(* Logix 5000 project; controller Safety vendor 1 type 14 code 148 rev 32.11; software revision 32.03; part 9 of 17 *)
(* tags used below, declared in another part *)
   DPD_EstopRstCmd : BOOL;   // DPD Estop Reset Cmd
   DPD_FltRstCmd : BOOL;   // DPD Fault Reset Cmd
   DPD_No_EStops : BOOL;   // DPD No Estops ( 1= OK)
   ESTOP_x281PB040 : DCI_STOP;   // OS9 Line EStop Pushbutton
   ESTOP_x281PB040_Flt : ALIAS FOR Flt_Estops.8;   // OS9 Line EStop Pushbutton Fault ( 1= Fault)
   ESTOP_x291PB040 : DCI_STOP;   // OS11 Line EStop Pushbutton
   ESTOP_x291PB040_Flt : ALIAS FOR Flt_Estops.9;   // OS11 Line EStop Pushbutton Fault ( 1= Fault)
   ESTOP_x301PB040 : DCI_STOP;   // OS13 Line EStop Pushbutton
   ESTOP_x301PB040_Flt : ALIAS FOR Flt_Estops.10;   // OS13 Line EStop Pushbutton Fault ( 1= Fault)
   ESTOP_x311PB040 : DCI_STOP;   // OS14 Line EStop Pushbutton
   ESTOP_x311PB040_Flt : ALIAS FOR Flt_Estops.11;   // OS14 Line EStop Pushbutton Fault ( 1= Fault)
   ESTOP_x321PB040 : DCI_STOP;   // OS15 Line EStop Pushbutton
   ESTOP_x321PB040_Flt : ALIAS FOR Flt_Estops.12;   // OS15 Line EStop Pushbutton Fault ( 1= Fault)
   ESTOP_x331PB040 : DCI_STOP;   // OS16 Line EStop Pushbutton
   ESTOP_x331PB040_Flt : ALIAS FOR Flt_Estops.13;   // OS16 Line EStop Pushbutton Fault ( 1= Fault)
   ESTOP_x480PB470 : DCI_STOP;   // DPD Line EStop Pushbutton
   ESTOP_x480PB470_Flt : ALIAS FOR Flt_Estops.14;   // DPD Line EStop Pushbutton Fault ( 1= Fault)
   ESTOP_x480PB550 : DCI_STOP;   // DPD (In Pit) Line EStop Pushbutton
   ESTOP_x480PB550_Flt : ALIAS FOR Flt_Estops.15;   // DPD Line EStop Pushbutton Fault ( 1= Fault)
   ESTOP_x519LS470 : DCI_STOP;   // G1 Tripwire Line EStop
   ESTOP_x519LS470_Flt : ALIAS FOR Flt_Estops.18;   // G1 Line EStop Tripwire Limit Switch Fault ( 1= Fault)
   ESTOP_x533PB470 : DCI_STOP;   // H1 Line EStop Pushbutton
   ESTOP_x533PB470_Flt : ALIAS FOR Flt_Estops.16;   // H1 Line EStop Pushbutton Fault ( 1= Fault)
   G1_EstopRstCmd : BOOL;   // G1 Estop Reset Command ( 1= Reset Cmd)
   G1_FltRstCmd : BOOL;   // G1 Fault Reset Command ( 1= Reset Cmd)
   G1_No_EStops : BOOL;   // G1 No Estops ( 1= OK)
   H1_EstopRstCmd : BOOL;   // H1 Estop Reset Command ( 1= Reset Cmd)
   H1_FltRstCmd : BOOL;   // H1 Fault Reset Command ( 1= Reset Cmd)
   H1_No_EStops : BOOL;   // H1 No Estops ( 1= OK)
   Line_TotalMode : BOOL;   // Line TOTAL Mode ( 1= Total Mode) (0 = Coil to Coil)
   LineSts : UDT_SysStatus;
   OS11_EstopRstCmd : BOOL;   // OS11 Estop Reset Command ( 1= Reset Cmd)
   OS11_FltRstCmd : BOOL;   // OS11 Fault Reset Command ( 1= Reset Cmd)
   OS11_No_EStops : BOOL;   // OS11 No Estops ( 1= OK)
   OS13_EstopRstCmd : BOOL;   // OS13 Estop Reset Command ( 1= Reset Cmd)
   OS13_FltRstCmd : BOOL;   // OS13 Fault Reset Command ( 1= Reset Cmd)
   OS13_No_EStops : BOOL;   // OS13 No Estops ( 1= OK)
   OS14_EstopRstCmd : BOOL;   // OS14 Estop Reset Command ( 1= Reset Cmd)
   OS14_FltRstCmd : BOOL;   // OS14 Fault Reset Command ( 1= Reset Cmd)
   OS14_No_EStops : BOOL;   // OS14 No Estops ( 1= OK)
   OS15_EstopRstCmd : BOOL;   // OS15 Estop Reset Command ( 1= Reset Cmd)
   OS15_FltRstCmd : BOOL;   // OS15 Fault Reset Command ( 1= Reset Cmd)
   OS15_No_EStops : BOOL;   // OS15 No Estops ( 1= OK)
   OS16_EstopRstCmd : BOOL;   // OS16 Estop Reset Command ( 1= Reset Cmd)
   OS16_FltRstCmd : BOOL;   // OS16 Fault Reset Command ( 1= Reset Cmd)
   OS16_No_EStops : BOOL;   // OS16 No Estops ( 1= OK)
   OS9_EstopRstCmd : BOOL;   // OS9 Estop Reset Command ( 1= Reset Cmd)
   OS9_FltRstCmd : BOOL;   // OS9 Fault Reset Command ( 1= Reset Cmd)
   OS9_No_EStops : BOOL;   // OS9 No Estops ( 1= OK)
   x281PB040a : ALIAS FOR OS9:1:I.Pt00Data;   // Emergency Stop PB
   x281PB040b : ALIAS FOR OS9:1:I.Pt01Data;   // Emergency Stop PB
   x291PB040a : ALIAS FOR OS11:1:I.Pt00Data;   // Emergency Stop PB
   x291PB040b : ALIAS FOR OS11:1:I.Pt01Data;   // Emergency Stop PB
   x301PB040a : ALIAS FOR OS13:1:I.Pt00Data;   // Emergency Stop PB
   x301PB040b : ALIAS FOR OS13:1:I.Pt01Data;   // Emergency Stop PB
   x311PB040a : ALIAS FOR OS14:1:I.Pt00Data;   // Emergency Stop PB OS14
   x311PB040b : ALIAS FOR OS14:1:I.Pt01Data;   // Emergency Stop PB OS14
   x321PB040a : ALIAS FOR OS15:1:I.Pt00Data;   // Emergency Stop PB
   x321PB040b : ALIAS FOR OS15:1:I.Pt01Data;   // Emergency Stop PB
   x331PB040a : ALIAS FOR OS16:1:I.Pt00Data;   // Emergency Stop PB
   x331PB040b : ALIAS FOR OS16:1:I.Pt01Data;   // Emergency Stop PB
   x480PB470a : ALIAS FOR DPD:15:I.Pt00Data;   // Emergency Stop Pushbutton
   x480PB470b : ALIAS FOR DPD:15:I.Pt01Data;   // Emergency Stop Pushbutton
   x480PB550a : ALIAS FOR DPD:15:I.Pt02Data;   // Emergency Stop Pushbutton (In Pit)
   x480PB550b : ALIAS FOR DPD:15:I.Pt03Data;   // Emergency Stop Pushbutton (In Pit)
   x519LS470 : ALIAS FOR G1:12:I.Pt00Data;   // Tripwire Emergency Stop Limit Switch
   x533PB470a : ALIAS FOR H1:6:I.Pt00Data;   // Sheeter Emergency Stop Pushbutton
   x533PB470b : ALIAS FOR H1:6:I.Pt01Data;   // Sheeter Emergency Stop Pushbutton
(* Estops, continued *)

ROUTINE A09_OS9_EStop   (* ladder *)
// OS9 EStops
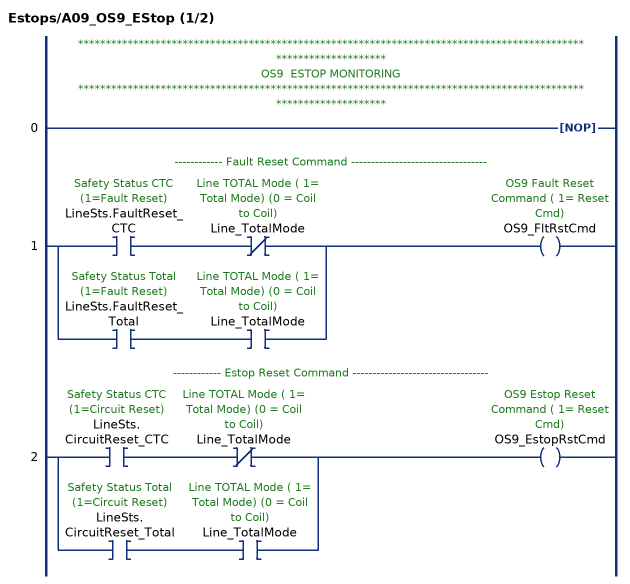
   // ****************************************************************************************************************
   // OS9  ESTOP MONITORING
   // ****************************************************************************************************************
   0: NOP();
   // ------------ Fault Reset Command ----------------------------------
   1: [XIC(LineSts.FaultReset_CTC) XIO(Line_TotalMode) ,XIC(LineSts.FaultReset_Total) XIC(Line_TotalMode) ]OTE(OS9_FltRstCmd);
   // ------------ Estop Reset Command ----------------------------------
   2: [XIC(LineSts.CircuitReset_CTC) XIO(Line_TotalMode) ,XIC(LineSts.CircuitReset_Total) XIC(Line_TotalMode) ]OTE(OS9_EstopRstCmd);
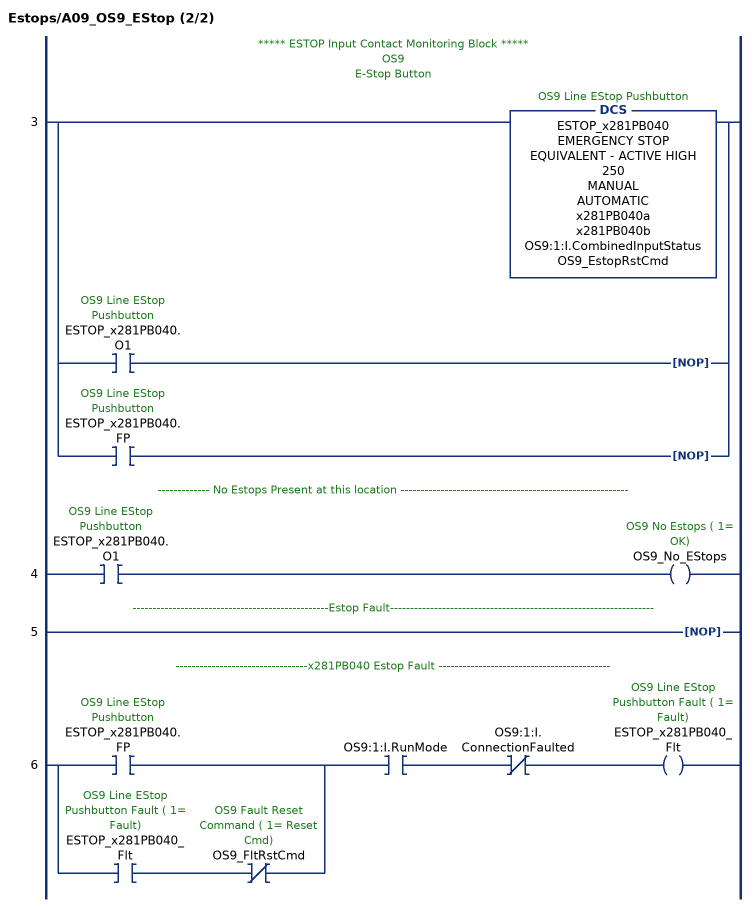
   // ***** ESTOP Input Contact Monitoring Block *****
   // OS9
   // E-Stop Button
   3: [DCS(ESTOP_x281PB040,EMERGENCY STOP,EQUIVALENT - ACTIVE HIGH,250,MANUAL,AUTOMATIC,x281PB040a,x281PB040b,OS9:1:I.CombinedInputStatus,OS9_EstopRstCmd) ,XIC(ESTOP_x281PB040.O1) NOP() ,XIC(ESTOP_x281PB040.FP) NOP() ];
   // ------------- No Estops Present at this location ---------------------------------------------------------
   4: XIC(ESTOP_x281PB040.O1)OTE(OS9_No_EStops);
   // -------------------------------------------------Estop Fault------------------------------------------------------------------
   5: NOP();
   // ---------------------------------x281PB040 Estop Fault -------------------------------------------
   6: [XIC(ESTOP_x281PB040.FP) ,XIC(ESTOP_x281PB040_Flt) XIO(OS9_FltRstCmd) ]XIC(OS9:1:I.RunMode)XIO(OS9:1:I.ConnectionFaulted)OTE(ESTOP_x281PB040_Flt);
END_ROUTINE

ROUTINE A11_OS11_EStop   (* ladder *)
// OS11 Estops
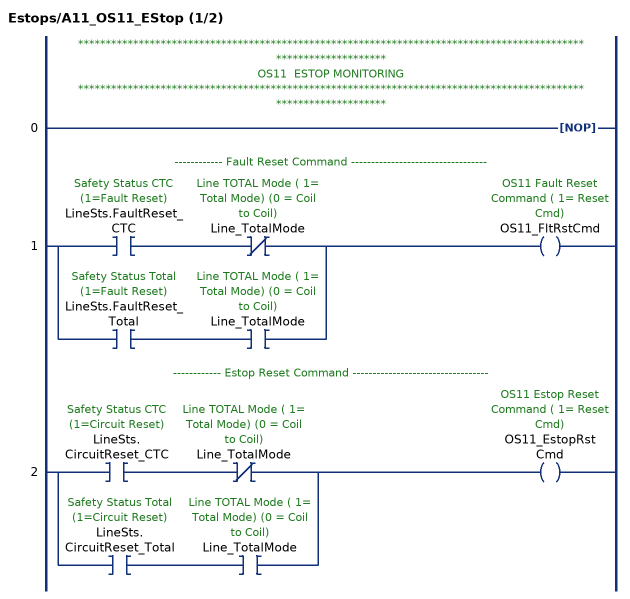
   // ****************************************************************************************************************
   // OS11  ESTOP MONITORING
   // ****************************************************************************************************************
   0: NOP();
   // ------------ Fault Reset Command ----------------------------------
   1: [XIC(LineSts.FaultReset_CTC) XIO(Line_TotalMode) ,XIC(LineSts.FaultReset_Total) XIC(Line_TotalMode) ]OTE(OS11_FltRstCmd);
   // ------------ Estop Reset Command ----------------------------------
   2: [XIC(LineSts.CircuitReset_CTC) XIO(Line_TotalMode) ,XIC(LineSts.CircuitReset_Total) XIC(Line_TotalMode) ]OTE(OS11_EstopRstCmd);
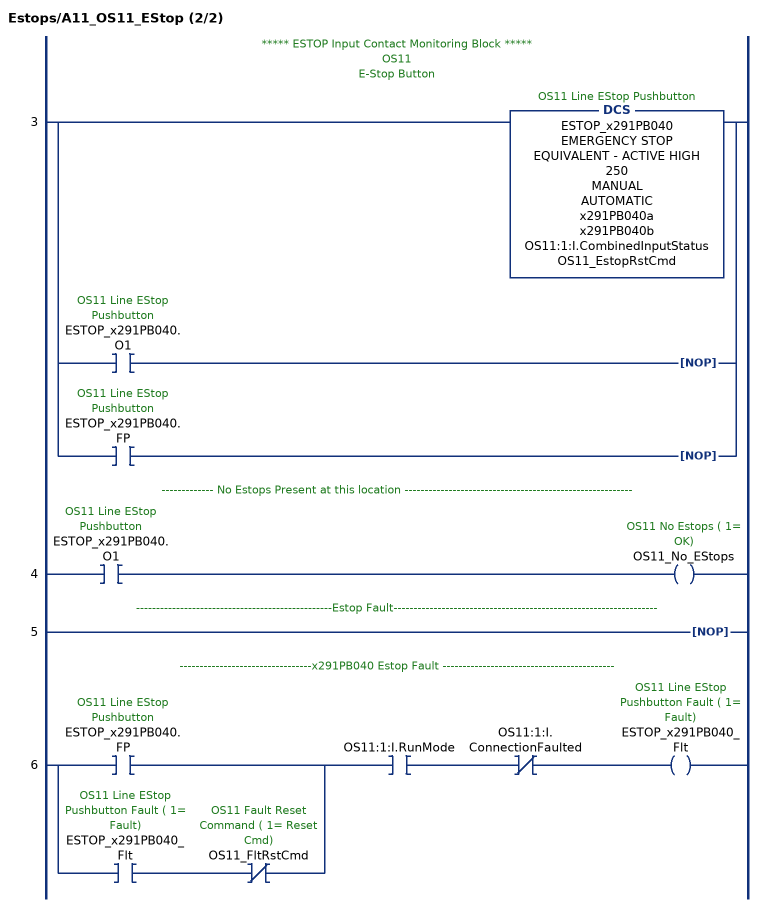
   // ***** ESTOP Input Contact Monitoring Block *****
   // OS11
   // E-Stop Button
   3: [DCS(ESTOP_x291PB040,EMERGENCY STOP,EQUIVALENT - ACTIVE HIGH,250,MANUAL,AUTOMATIC,x291PB040a,x291PB040b,OS11:1:I.CombinedInputStatus,OS11_EstopRstCmd) ,XIC(ESTOP_x291PB040.O1) NOP() ,XIC(ESTOP_x291PB040.FP) NOP() ];
   // ------------- No Estops Present at this location ---------------------------------------------------------
   4: XIC(ESTOP_x291PB040.O1)OTE(OS11_No_EStops);
   // -------------------------------------------------Estop Fault------------------------------------------------------------------
   5: NOP();
   // ---------------------------------x291PB040 Estop Fault -------------------------------------------
   6: [XIC(ESTOP_x291PB040.FP) ,XIC(ESTOP_x291PB040_Flt) XIO(OS11_FltRstCmd) ]XIC(OS11:1:I.RunMode)XIO(OS11:1:I.ConnectionFaulted)OTE(ESTOP_x291PB040_Flt);
END_ROUTINE

ROUTINE A13_OS13_EStop   (* ladder *)
// OS13 EStops
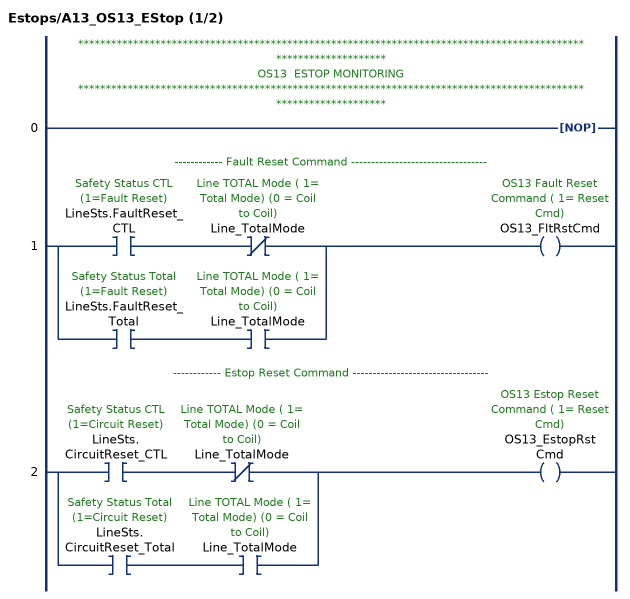
   // ****************************************************************************************************************
   // OS13  ESTOP MONITORING
   // ****************************************************************************************************************
   0: NOP();
   // ------------ Fault Reset Command ----------------------------------
   1: [XIC(LineSts.FaultReset_CTL) XIO(Line_TotalMode) ,XIC(LineSts.FaultReset_Total) XIC(Line_TotalMode) ]OTE(OS13_FltRstCmd);
   // ------------ Estop Reset Command ----------------------------------
   2: [XIC(LineSts.CircuitReset_CTL) XIO(Line_TotalMode) ,XIC(LineSts.CircuitReset_Total) XIC(Line_TotalMode) ]OTE(OS13_EstopRstCmd);
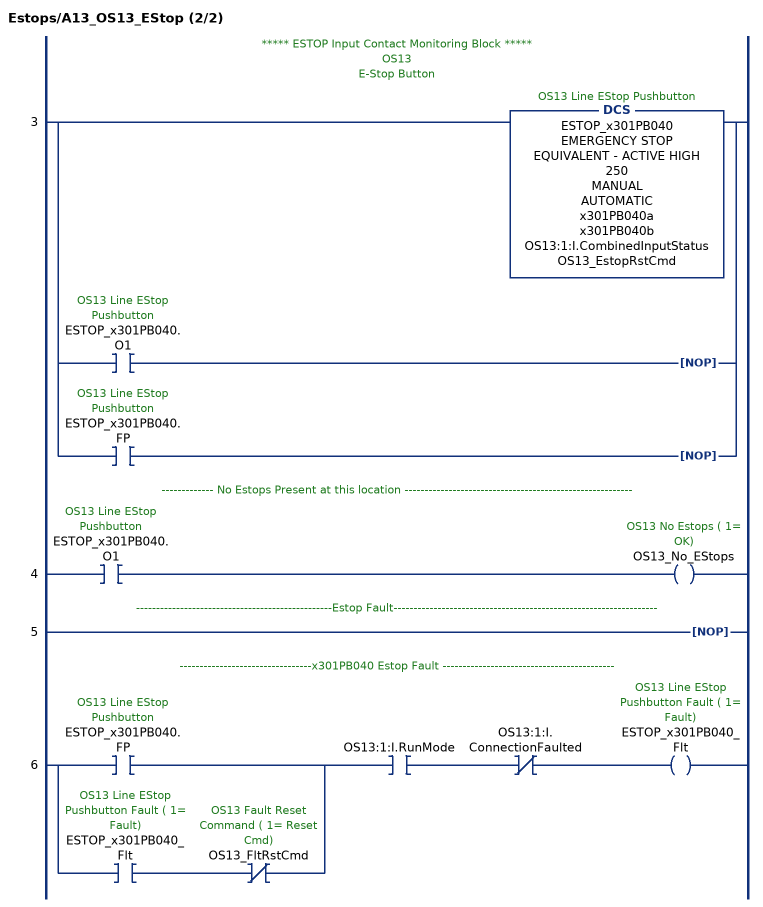
   // ***** ESTOP Input Contact Monitoring Block *****
   // OS13
   // E-Stop Button
   3: [DCS(ESTOP_x301PB040,EMERGENCY STOP,EQUIVALENT - ACTIVE HIGH,250,MANUAL,AUTOMATIC,x301PB040a,x301PB040b,OS13:1:I.CombinedInputStatus,OS13_EstopRstCmd) ,XIC(ESTOP_x301PB040.O1) NOP() ,XIC(ESTOP_x301PB040.FP) NOP() ];
   // ------------- No Estops Present at this location ---------------------------------------------------------
   4: XIC(ESTOP_x301PB040.O1)OTE(OS13_No_EStops);
   // -------------------------------------------------Estop Fault------------------------------------------------------------------
   5: NOP();
   // ---------------------------------x301PB040 Estop Fault -------------------------------------------
   6: [XIC(ESTOP_x301PB040.FP) ,XIC(ESTOP_x301PB040_Flt) XIO(OS13_FltRstCmd) ]XIC(OS13:1:I.RunMode)XIO(OS13:1:I.ConnectionFaulted)OTE(ESTOP_x301PB040_Flt);
END_ROUTINE

ROUTINE A14_OS14_EStop   (* ladder *)
// OS14 EStop
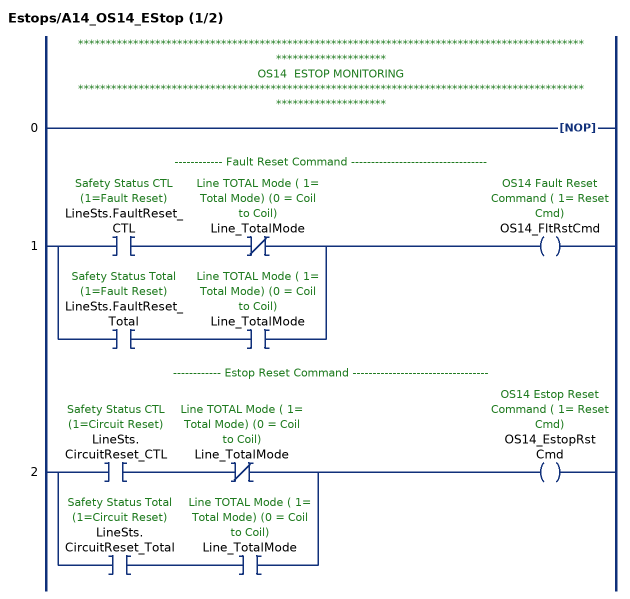
   // ****************************************************************************************************************
   // OS14  ESTOP MONITORING
   // ****************************************************************************************************************
   0: NOP();
   // ------------ Fault Reset Command ----------------------------------
   1: [XIC(LineSts.FaultReset_CTL) XIO(Line_TotalMode) ,XIC(LineSts.FaultReset_Total) XIC(Line_TotalMode) ]OTE(OS14_FltRstCmd);
   // ------------ Estop Reset Command ----------------------------------
   2: [XIC(LineSts.CircuitReset_CTL) XIO(Line_TotalMode) ,XIC(LineSts.CircuitReset_Total) XIC(Line_TotalMode) ]OTE(OS14_EstopRstCmd);
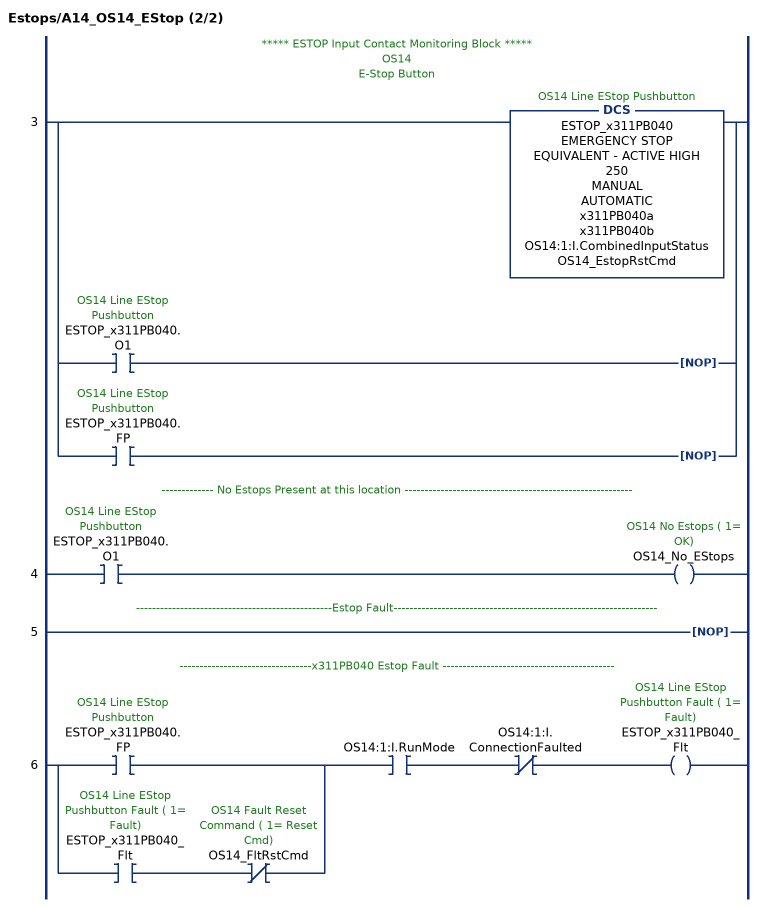
   // ***** ESTOP Input Contact Monitoring Block *****
   // OS14
   // E-Stop Button
   3: [DCS(ESTOP_x311PB040,EMERGENCY STOP,EQUIVALENT - ACTIVE HIGH,250,MANUAL,AUTOMATIC,x311PB040a,x311PB040b,OS14:1:I.CombinedInputStatus,OS14_EstopRstCmd) ,XIC(ESTOP_x311PB040.O1) NOP() ,XIC(ESTOP_x311PB040.FP) NOP() ];
   // ------------- No Estops Present at this location ---------------------------------------------------------
   4: XIC(ESTOP_x311PB040.O1)OTE(OS14_No_EStops);
   // -------------------------------------------------Estop Fault------------------------------------------------------------------
   5: NOP();
   // ---------------------------------x311PB040 Estop Fault -------------------------------------------
   6: [XIC(ESTOP_x311PB040.FP) ,XIC(ESTOP_x311PB040_Flt) XIO(OS14_FltRstCmd) ]XIC(OS14:1:I.RunMode)XIO(OS14:1:I.ConnectionFaulted)OTE(ESTOP_x311PB040_Flt);
END_ROUTINE

ROUTINE A15_OS15_EStop   (* ladder *)
// OS15 EStops
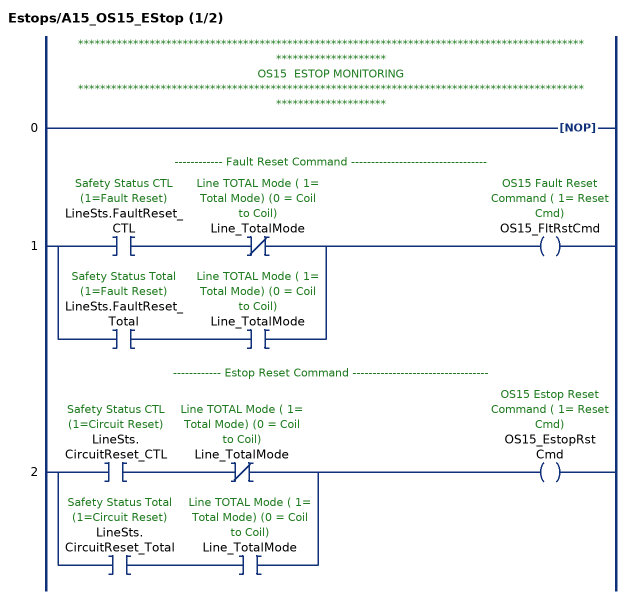
   // ****************************************************************************************************************
   // OS15  ESTOP MONITORING
   // ****************************************************************************************************************
   0: NOP();
   // ------------ Fault Reset Command ----------------------------------
   1: [XIC(LineSts.FaultReset_CTL) XIO(Line_TotalMode) ,XIC(LineSts.FaultReset_Total) XIC(Line_TotalMode) ]OTE(OS15_FltRstCmd);
   // ------------ Estop Reset Command ----------------------------------
   2: [XIC(LineSts.CircuitReset_CTL) XIO(Line_TotalMode) ,XIC(LineSts.CircuitReset_Total) XIC(Line_TotalMode) ]OTE(OS15_EstopRstCmd);
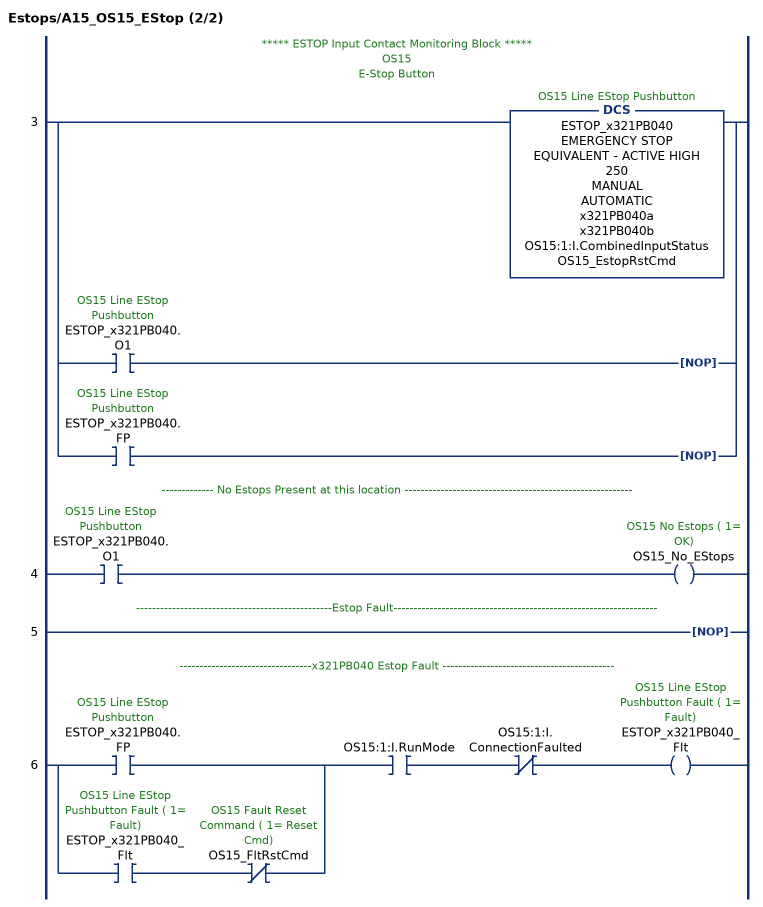
   // ***** ESTOP Input Contact Monitoring Block *****
   // OS15
   // E-Stop Button
   3: [DCS(ESTOP_x321PB040,EMERGENCY STOP,EQUIVALENT - ACTIVE HIGH,250,MANUAL,AUTOMATIC,x321PB040a,x321PB040b,OS15:1:I.CombinedInputStatus,OS15_EstopRstCmd) ,XIC(ESTOP_x321PB040.O1) NOP() ,XIC(ESTOP_x321PB040.FP) NOP() ];
   // ------------- No Estops Present at this location ---------------------------------------------------------
   4: XIC(ESTOP_x321PB040.O1)OTE(OS15_No_EStops);
   // -------------------------------------------------Estop Fault------------------------------------------------------------------
   5: NOP();
   // ---------------------------------x321PB040 Estop Fault -------------------------------------------
   6: [XIC(ESTOP_x321PB040.FP) ,XIC(ESTOP_x321PB040_Flt) XIO(OS15_FltRstCmd) ]XIC(OS15:1:I.RunMode)XIO(OS15:1:I.ConnectionFaulted)OTE(ESTOP_x321PB040_Flt);
END_ROUTINE

ROUTINE A16_OS16_EStop   (* ladder *)
// OS16 EStops
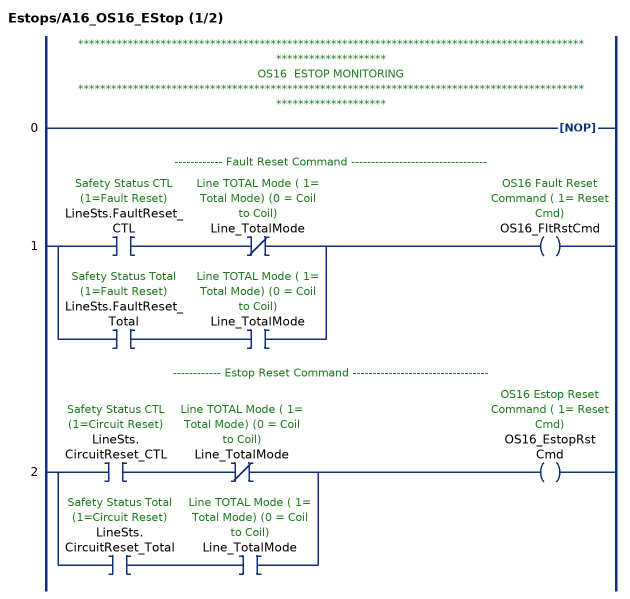
   // ****************************************************************************************************************
   // OS16  ESTOP MONITORING
   // ****************************************************************************************************************
   0: NOP();
   // ------------ Fault Reset Command ----------------------------------
   1: [XIC(LineSts.FaultReset_CTL) XIO(Line_TotalMode) ,XIC(LineSts.FaultReset_Total) XIC(Line_TotalMode) ]OTE(OS16_FltRstCmd);
   // ------------ Estop Reset Command ----------------------------------
   2: [XIC(LineSts.CircuitReset_CTL) XIO(Line_TotalMode) ,XIC(LineSts.CircuitReset_Total) XIC(Line_TotalMode) ]OTE(OS16_EstopRstCmd);
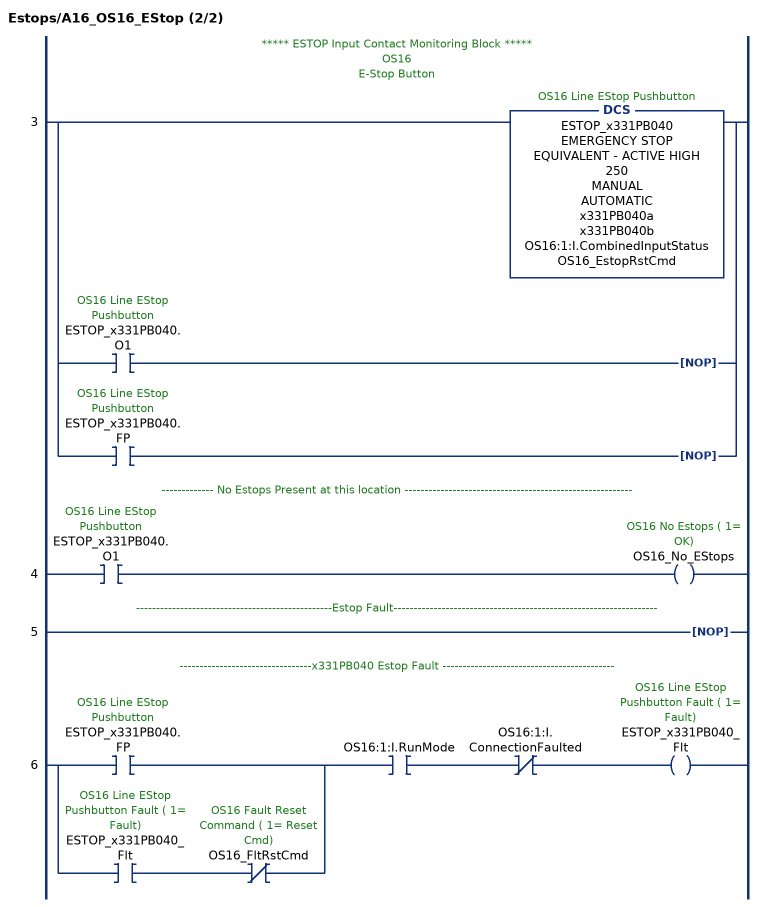
   // ***** ESTOP Input Contact Monitoring Block *****
   // OS16
   // E-Stop Button
   3: [DCS(ESTOP_x331PB040,EMERGENCY STOP,EQUIVALENT - ACTIVE HIGH,250,MANUAL,AUTOMATIC,x331PB040a,x331PB040b,OS16:1:I.CombinedInputStatus,OS16_EstopRstCmd) ,XIC(ESTOP_x331PB040.O1) NOP() ,XIC(ESTOP_x331PB040.FP) NOP() ];
   // ------------- No Estops Present at this location ---------------------------------------------------------
   4: XIC(ESTOP_x331PB040.O1)OTE(OS16_No_EStops);
   // -------------------------------------------------Estop Fault------------------------------------------------------------------
   5: NOP();
   // ---------------------------------x331PB040 Estop Fault -------------------------------------------
   6: [XIC(ESTOP_x331PB040.FP) ,XIC(ESTOP_x331PB040_Flt) XIO(OS16_FltRstCmd) ]XIC(OS16:1:I.RunMode)XIO(OS16:1:I.ConnectionFaulted)OTE(ESTOP_x331PB040_Flt);
END_ROUTINE

ROUTINE B00_DPD_Estop   (* ladder *)
// DPD IO Panel EStop
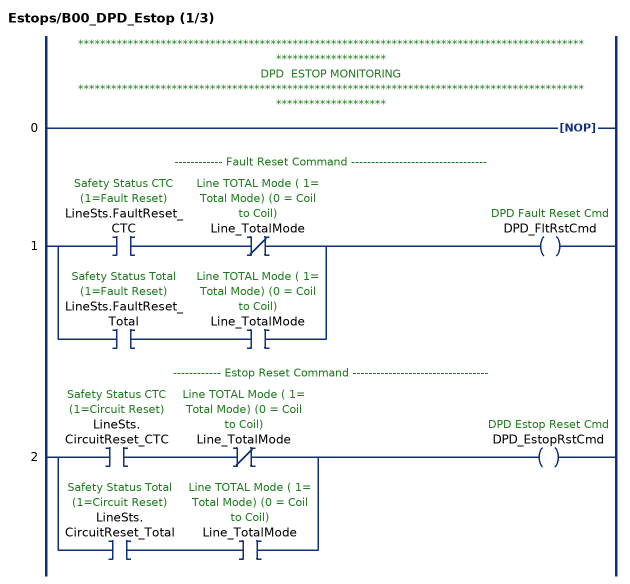
   // ****************************************************************************************************************
   // DPD  ESTOP MONITORING
   // ****************************************************************************************************************
   0: NOP();
   // ------------ Fault Reset Command ----------------------------------
   1: [XIC(LineSts.FaultReset_CTC) XIO(Line_TotalMode) ,XIC(LineSts.FaultReset_Total) XIC(Line_TotalMode) ]OTE(DPD_FltRstCmd);
   // ------------ Estop Reset Command ----------------------------------
   2: [XIC(LineSts.CircuitReset_CTC) XIO(Line_TotalMode) ,XIC(LineSts.CircuitReset_Total) XIC(Line_TotalMode) ]OTE(DPD_EstopRstCmd);
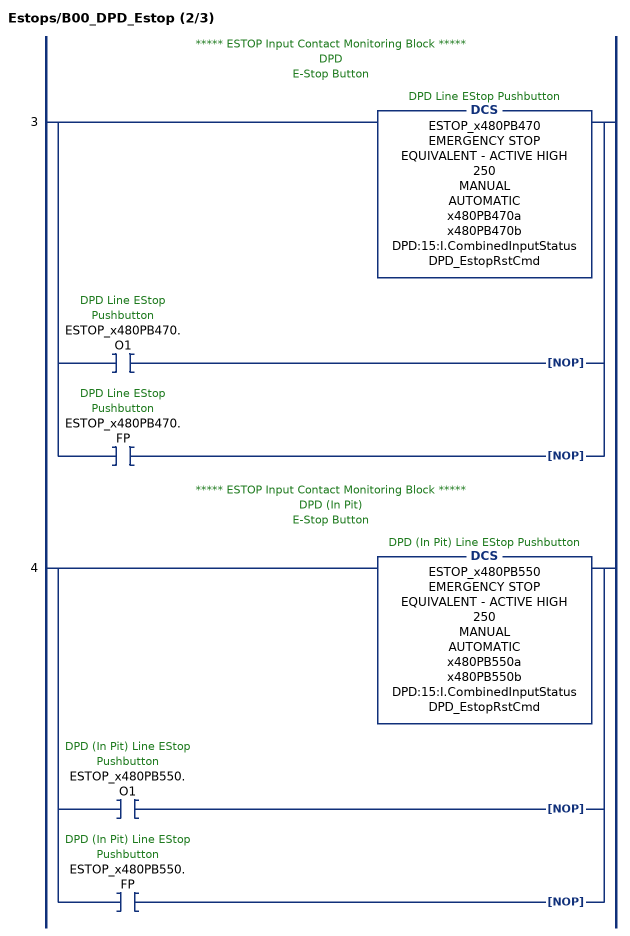
   // ***** ESTOP Input Contact Monitoring Block *****
   // DPD
   // E-Stop Button
   3: [DCS(ESTOP_x480PB470,EMERGENCY STOP,EQUIVALENT - ACTIVE HIGH,250,MANUAL,AUTOMATIC,x480PB470a,x480PB470b,DPD:15:I.CombinedInputStatus,DPD_EstopRstCmd) ,XIC(ESTOP_x480PB470.O1) NOP() ,XIC(ESTOP_x480PB470.FP) NOP() ];
   // ***** ESTOP Input Contact Monitoring Block *****
   // DPD (In Pit)
   // E-Stop Button
   4: [DCS(ESTOP_x480PB550,EMERGENCY STOP,EQUIVALENT - ACTIVE HIGH,250,MANUAL,AUTOMATIC,x480PB550a,x480PB550b,DPD:15:I.CombinedInputStatus,DPD_EstopRstCmd) ,XIC(ESTOP_x480PB550.O1) NOP() ,XIC(ESTOP_x480PB550.FP) NOP() ];
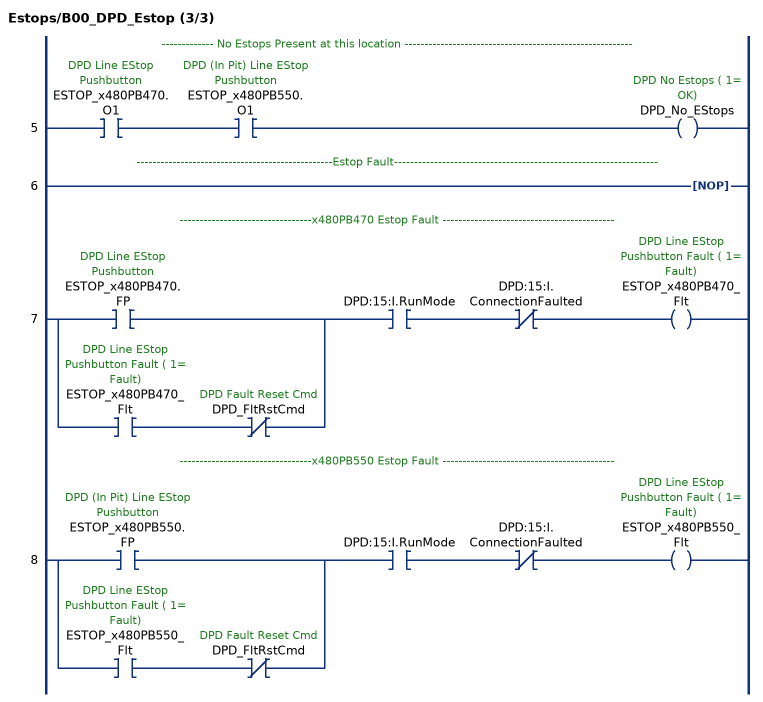
   // ------------- No Estops Present at this location ---------------------------------------------------------
   5: XIC(ESTOP_x480PB470.O1)XIC(ESTOP_x480PB550.O1)OTE(DPD_No_EStops);
   // -------------------------------------------------Estop Fault------------------------------------------------------------------
   6: NOP();
   // ---------------------------------x480PB470 Estop Fault -------------------------------------------
   7: [XIC(ESTOP_x480PB470.FP) ,XIC(ESTOP_x480PB470_Flt) XIO(DPD_FltRstCmd) ]XIC(DPD:15:I.RunMode)XIO(DPD:15:I.ConnectionFaulted)OTE(ESTOP_x480PB470_Flt);
   // ---------------------------------x480PB550 Estop Fault -------------------------------------------
   8: [XIC(ESTOP_x480PB550.FP) ,XIC(ESTOP_x480PB550_Flt) XIO(DPD_FltRstCmd) ]XIC(DPD:15:I.RunMode)XIO(DPD:15:I.ConnectionFaulted)OTE(ESTOP_x480PB550_Flt);
END_ROUTINE

ROUTINE B01_H1_EStop   (* ladder *)
// H1 IO Panel Estop
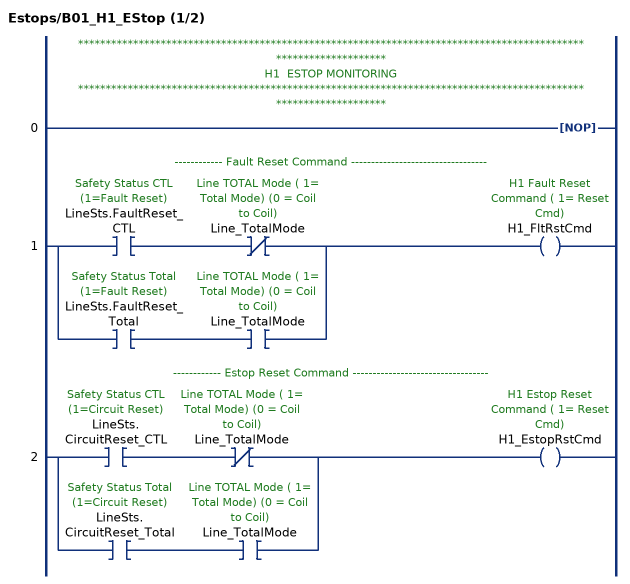
   // ****************************************************************************************************************
   // H1  ESTOP MONITORING
   // ****************************************************************************************************************
   0: NOP();
   // ------------ Fault Reset Command ----------------------------------
   1: [XIC(LineSts.FaultReset_CTL) XIO(Line_TotalMode) ,XIC(LineSts.FaultReset_Total) XIC(Line_TotalMode) ]OTE(H1_FltRstCmd);
   // ------------ Estop Reset Command ----------------------------------
   2: [XIC(LineSts.CircuitReset_CTL) XIO(Line_TotalMode) ,XIC(LineSts.CircuitReset_Total) XIC(Line_TotalMode) ]OTE(H1_EstopRstCmd);
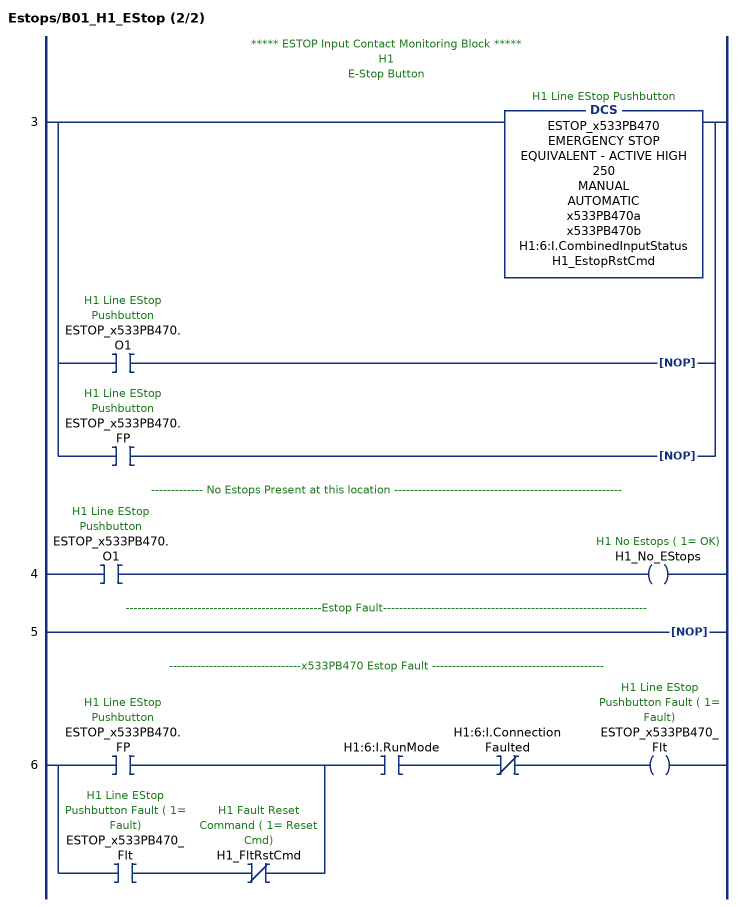
   // ***** ESTOP Input Contact Monitoring Block *****
   // H1
   // E-Stop Button
   3: [DCS(ESTOP_x533PB470,EMERGENCY STOP,EQUIVALENT - ACTIVE HIGH,250,MANUAL,AUTOMATIC,x533PB470a,x533PB470b,H1:6:I.CombinedInputStatus,H1_EstopRstCmd) ,XIC(ESTOP_x533PB470.O1) NOP() ,XIC(ESTOP_x533PB470.FP) NOP() ];
   // ------------- No Estops Present at this location ---------------------------------------------------------
   4: XIC(ESTOP_x533PB470.O1)OTE(H1_No_EStops);
   // -------------------------------------------------Estop Fault------------------------------------------------------------------
   5: NOP();
   // ---------------------------------x533PB470 Estop Fault -------------------------------------------
   6: [XIC(ESTOP_x533PB470.FP) ,XIC(ESTOP_x533PB470_Flt) XIO(H1_FltRstCmd) ]XIC(H1:6:I.RunMode)XIO(H1:6:I.ConnectionFaulted)OTE(ESTOP_x533PB470_Flt);
END_ROUTINE

ROUTINE B02_G1_EStop   (* ladder *)
// G1 IO Panel Estop
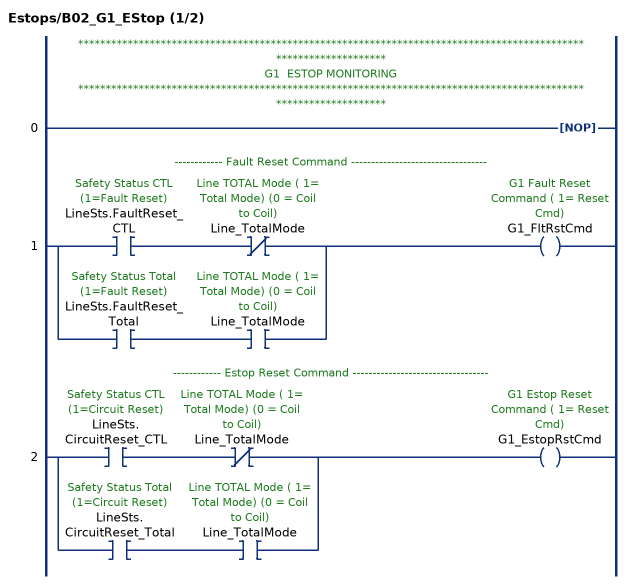
   // ****************************************************************************************************************
   // G1  ESTOP MONITORING
   // ****************************************************************************************************************
   0: NOP();
   // ------------ Fault Reset Command ----------------------------------
   1: [XIC(LineSts.FaultReset_CTL) XIO(Line_TotalMode) ,XIC(LineSts.FaultReset_Total) XIC(Line_TotalMode) ]OTE(G1_FltRstCmd);
   // ------------ Estop Reset Command ----------------------------------
   2: [XIC(LineSts.CircuitReset_CTL) XIO(Line_TotalMode) ,XIC(LineSts.CircuitReset_Total) XIC(Line_TotalMode) ]OTE(G1_EstopRstCmd);
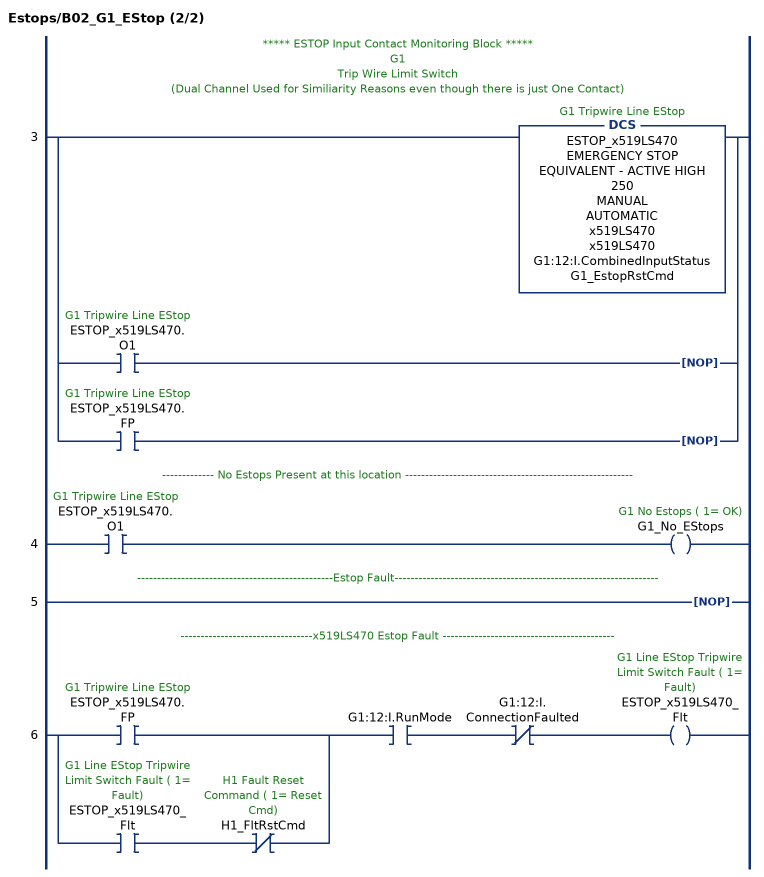
   // ***** ESTOP Input Contact Monitoring Block *****
   // G1
   // Trip Wire Limit Switch
   // (Dual Channel Used for Similiarity Reasons even though there is just One Contact)
   3: [DCS(ESTOP_x519LS470,EMERGENCY STOP,EQUIVALENT - ACTIVE HIGH,250,MANUAL,AUTOMATIC,x519LS470,x519LS470,G1:12:I.CombinedInputStatus,G1_EstopRstCmd) ,XIC(ESTOP_x519LS470.O1) NOP() ,XIC(ESTOP_x519LS470.FP) NOP() ];
   // ------------- No Estops Present at this location ---------------------------------------------------------
   4: XIC(ESTOP_x519LS470.O1)OTE(G1_No_EStops);
   // -------------------------------------------------Estop Fault------------------------------------------------------------------
   5: NOP();
   // ---------------------------------x519LS470 Estop Fault -------------------------------------------
   6: [XIC(ESTOP_x519LS470.FP) ,XIC(ESTOP_x519LS470_Flt) XIO(H1_FltRstCmd) ]XIC(G1:12:I.RunMode)XIO(G1:12:I.ConnectionFaulted)OTE(ESTOP_x519LS470_Flt);
END_ROUTINE
